(* CODESYS project zamek.project

Project tree, tasks and I/O mapping:
  Device : CODESYS Control Win V3, 3S - Smart Software Solutions GmbH, order no. 305021, version 3.5.8.10
    application Application
      libraries: Standard, * (System)
      task MainTask (cyclic, interval t#20ms, priority 1) calls PLC_PRG
      task VISU_TASK (cyclic, interval 100 ms, priority 31) calls VisuElems.Visu_Prg
      program PLC_PRG [ST]
      visualisation Visualization
  libraries: VisuSymbols, 3.5.8.0 (System)
  text list GlobalTextList
*)

// Device/Application/PLC_PRG
PROGRAM PLC_PRG

VAR								// Początek sekcji zmiennych
	
	xPrzycisk0: BOOL := FALSE;		// Zmienna stanu przycisku z cyfrą 0 (typ przycisku "pushswitch")	-> Zainicjalizowana wartością "false"
	xPrzycisk1: BOOL := FALSE;		// Zmienna stanu przycisku z cyfrą 1 (typ przycisku "pushswitch")	-> Zainicjalizowana wartością "false"	
	xPrzycisk2: BOOL := FALSE;		// Zmienna stanu przycisku z cyfrą 2 (typ przycisku "pushswitch")	-> Zainicjalizowana wartością "false"	
	xPrzycisk3: BOOL := FALSE;		// Zmienna stanu przycisku z cyfrą 3 (typ przycisku "pushswitch")	-> Zainicjalizowana wartością "false"	
	xPrzycisk4: BOOL := FALSE;		// Zmienna stanu przycisku z cyfrą 4 (typ przycisku "pushswitch")	-> Zainicjalizowana wartością "false"	
	xPrzycisk5: BOOL := FALSE;		// Zmienna stanu przycisku z cyfrą 5 (typ przycisku "pushswitch")	-> Zainicjalizowana wartością "false"	
	xPrzycisk6: BOOL := FALSE;		// Zmienna stanu przycisku z cyfrą 6 (typ przycisku "pushswitch")	-> Zainicjalizowana wartością "false"	
	xPrzycisk7: BOOL := FALSE;		// Zmienna stanu przycisku z cyfrą 7 (typ przycisku "pushswitch")	-> Zainicjalizowana wartością "false"	
	xPrzycisk8: BOOL := FALSE;		// Zmienna stanu przycisku z cyfrą 8 (typ przycisku "pushswitch")	-> Zainicjalizowana wartością "false"	
	xPrzycisk9: BOOL := FALSE;		// Zmienna stanu przycisku z cyfrą 9 (typ przycisku "pushswitch")	-> Zainicjalizowana wartością "false"	
	
	xKlucz: BOOL;					// Zmienna stanu przycisku typu "PowerSwitch" o nazwie "klucz"	
	xLampka1: BOOL;					// Zmienna oznaczająca stan lampki zielonej (typ "lamp1") - zapala się po wprowadzeniu prawidłowej sekwencji 4 cyfr
	xLampka2: BOOL;					// Zmienna oznaczająca stan lampki czerwonej (typ "lamp1") - zapala się po wprowadzeniu nieprawidłowej sekwencji cyfr
	
	xSpr1: BOOL;					// Zmienna typu "BOOL" oznaczająca wystukanie pierwszej poprawnej cyfry
	xSpr2: BOOL;					// Zmienna typu "BOOL" oznaczająca wystukanie drugiej poprawnej cyfry (1 cyfra poprawna musi być wprowadzona) 
	xSpr3: BOOL;					// Zmienna typu "BOOL" oznaczająca wystukanie trzeciej poprawnej cyfry (1 i 2 cyfra poprawna muszą być wprowadzone) 
	xSpr4: BOOL;					// Zmienna typu "BOOL" oznaczająca wystukanie czwartej poprawnej cyfry (1 i 2 i 3 cyfra poprawna muszą być wprowadzone)

	xOdblokuj: BOOL;				// Zmienna true/false zapalająca się (stan wysoki) jeśli cyfry poprawne zostały wprowadzone w prawidłowej sekwencji oraz oprócz tego czy przycisk "xKlucz" jest aktywny
	T3: TON;						// Deklaracja bloku funkcji Timer on-delay, który przeprowadza opóźnienie załączania stanu wysokiego w zmiennej "xOdblokuj2". Wynika z przyjętego algorytmu - ustawione opóźnienie jest niezauważalne
	xOdblokuj2: BOOL;				// Zmienna przyjmująca stan wysoki po upływie 1ms od ustawienia stanu wyokiego na zmiennej xOdblokuj 
	T1: TOF;						// Deklaracja bloku funkcji Timer off-delay przeprowadzającego opóźnienie wyłączenia lampki zielonej (xLampka1) - po 5s. Startuje swoje działanie, jeżeli zmienna xOdblokuj osiągnie opadające zbocze
	
	xNieOdblokuj: BOOL;				// Zmienna do obsługi wprowadzonego nieprawidłowego kodu / sekwencji. Osiąga stan wysoki jeżeli xKlucz osiąga stan wysoki, ale któraś ze zmiennych spr1,spr2,spr3,spr4 ma ustawiony stan niski
	T4: TON;						// Timer opóżniający zapalenie stanu wysokiego na zmiennej xNieOdblokuj2 o 1ms. Wynika z przyjętego algorytmu - ustawione opóźnienie jest niezauważalne.
	xNieOdblokuj2: BOOL;			// Zapala sie poprzez Timer po upłynięciu 1ms stanu wysokiego na zmiennej xNieOdblokuj		
	T2: TOF;						// Timer, który przy stanie niski zmiennej xNieOdblokuj załącza lampke czerwoną na 10s
	

	xNieaktywny: BOOL := FALSE;		// Zmienna służąca do poinformowaniu o bezczynności przycisku 'klucz' jeżeli któraś z lampek jest zapalona. Jest pezpośrednio podłączona do "xKlucz" powershitch do wejścia "deactivate inputs" w wizualizacji (powerswitch properties)
	
	xLicznikProb1: INT := 0;		// Licznik nieudanych prób. Jest zwiększany o 2 przy każdej nieudanej próbie (przy sprawdzaniu spr1,spr2,spr3,spr4 oraz zKlucz). Kiedy osiąga wartość 6 - 3 nieudane próby - następuje załączenie lampki czerwonej na 3min.
	
	xBlokuj: BOOL := FALSE;			// Jest odpowiednikiem xNieOdblokuj - stworzona w celu obsługi trzyminutowego zapalenia czerwonej lampki. Stworzona na potrzeby przyjętego algorytmu - 'steruje' zmienną xBlokuj2
	xBlokuj2: BOOL := FALSE;		// Jest odpowiednikiem xNieOdblokuj2 - stworzona w celu obsługi trzyminutowego zapalenia czerwonej lampki. Jej stan niski powoduje opóźnienie (zapalenia lampki czerwonej) na 3min
	
	T5: TOF;						// Odpowiednik Timera T2, który odpowiada za bezpośrednie ustawienie stanu wysokiego na lampce czerwonej na 3min
	T6: TON;						// Odpowiednik Timera T4, który po upływie 1ms ustawia stan niski na xBlokuj2
	
	xZerujLIcznik2: BOOL := FALSE;	// Zmienna stworzona do sprawdzania liczby prób (xLiczbProb1). Przyjmuje stan wysoki jeżeli 3 próba z kolei się nie powiodła 
	xZerujLIcznik: BOOL := FALSE;	// Zapala się tutaj stan wysoki po upłynięciu 3 min od zapalenia stanu wysokiego na zmiennej xZerujLicznik2. Te dwie zmienne sterują prawidłowym procesem zerowania liczby prób po upływie 3 minut - 3 nieudane próby
	T7: TON;						// Blok Timer, który ustawia stan wysoki na zmiennej xZerujLIcznik po upłynięciu 3 min ustawienia lampki czerwonej - stanu wysokiego na zmiennej xZerujLicznik2
	
END_VAR							// Koniec sekcji zmiennych

// Sekcja właściwego kodu programu

	// KOD POPRAWNY DO OTWORZENIA ZAMKA: 1234
	// KOD POPRAWNY DO OTWORZENIA ZAMKA: 1234
	// KOD POPRAWNY DO OTWORZENIA ZAMKA: 1234
	
	// Sprawdzanie prawidłowej sekwencji oraz prawidłowych cyfr zamka
	
		// Czy przycisk z cyfrą 1 został naciśnięty - żadne inne
		
			IF (xPrzycisk0=FALSE AND xPrzycisk5=FALSE AND xPrzycisk6=FALSE AND xPrzycisk7=FALSE AND xPrzycisk8=FALSE AND xPrzycisk9=FALSE) AND xPrzycisk1=TRUE AND xPrzycisk2=FALSE AND xPrzycisk3=FALSE AND xPrzycisk4=FALSE AND xKlucz=FALSE THEN
				xSpr1:=TRUE;
			END_IF

		// Czy przycisk z cyfrą 2 został naciśnięty (i przycisk z cyfrą 1 jest dalej aktywny) - żadne inne
			
			IF (xPrzycisk0=FALSE AND xPrzycisk5=FALSE AND xPrzycisk6=FALSE AND xPrzycisk7=FALSE AND xPrzycisk8=FALSE AND xPrzycisk9=FALSE) AND xPrzycisk2=TRUE AND xPrzycisk3=FALSE AND xPrzycisk4=FALSE AND xSpr1=TRUE AND xKlucz=FALSE THEN
				xSpr2:=TRUE;
			END_IF
			
		// Czy przycisk z cyfrą 3 został naciśnięty (i przycisk z cyfrą 1 i 2 jest dalej aktywny) - żadne inne

			IF (xPrzycisk0=FALSE AND xPrzycisk5=FALSE AND xPrzycisk6=FALSE AND xPrzycisk7=FALSE AND xPrzycisk8=FALSE AND xPrzycisk9=FALSE) AND xPrzycisk3=TRUE AND xPrzycisk4=FALSE AND xSpr1=TRUE AND xSpr2=TRUE AND xKlucz=FALSE THEN
				xSpr3:=TRUE;
			END_IF
			
		// Jeżeli został wciśnięty inny przycisk to zmienna określająca wysoki stan na przycisku 1 2 3 zmienia się na false - zapobiegnięcie m.in. sytuacji kodu 1 2 3 4 5

			IF (xPrzycisk5=TRUE OR xPrzycisk6=TRUE OR xPrzycisk7=TRUE OR xPrzycisk8=TRUE OR xPrzycisk9=TRUE) THEN
				xSpr3:=FALSE;
			END_IF
			
		// Czy przycisk z cyfrą 4 został naciśnięty (i przycisk z cyfrą 1 i 2 i 3 jest dalej aktywny) - żadne inne

			IF (xPrzycisk0=FALSE AND xPrzycisk5=FALSE AND xPrzycisk6=FALSE AND xPrzycisk7=FALSE AND xPrzycisk8=FALSE AND xPrzycisk9=FALSE) AND xPrzycisk4=TRUE AND xSpr1=TRUE AND xSpr2=TRUE AND xSpr3=TRUE AND xKlucz=FALSE THEN
				xSpr4:=TRUE;
			END_IF
		
		// Sekwencja 1 2 3 4 ustawia stan wysoki na zmiennej xOdblokuj (zaraz po naciśnięciu przycisku klucz)
			
			IF xSpr1=TRUE AND xSpr2=TRUE AND xSpr3=TRUE AND xSpr4=TRUE AND xKlucz=TRUE THEN
				xOdblokuj:=TRUE;
			END_IF

		// Kod wynikający z opracowanego algorytmu. Zmiana stanu zmainnej xOdblokuj2 (na wysoki) pod wpływem ustawienia stanu wysokiego xOdblokuj po 1ms 	
			
			T3(IN:=xOdblokuj,PT:=T#1MS);		// Deklaracja Timera TON. IN-zmienna wejściowa, PT-czas do ustawienia zmiennej wyjściowej
			xOdblokuj2:=T3.Q;					// Poinformowanie o zmiennej wyjściowej

		// Kod poniżej wykouje się w przypadku prawidłowej sekwencji. Wszystkie potrzebne przyciski, zmienne sprawdzające, licznik nieudanych prób, zostają "zresetowane" - ustawione na stan niski	
			
			IF xOdblokuj2=TRUE THEN
				xOdblokuj:=FALSE;
				
				xSpr1:=FALSE;
				xSpr2:=FALSE;
				xSpr3:=FALSE;
				xSpr4:=FALSE;
				
				xKlucz:=FALSE;
				xPrzycisk0:=FALSE;	
				xPrzycisk1:=FALSE;	
				xPrzycisk2:=FALSE;
				xPrzycisk3:=FALSE;
				xPrzycisk4:=FALSE;
				xPrzycisk5:=FALSE;
				xPrzycisk6:=FALSE;
				xPrzycisk7:=FALSE;
				xPrzycisk8:=FALSE;
				xPrzycisk9:=FALSE;
				
				xBlokuj:=FALSE;
				xBlokuj2:=FALSE;
				
				xLicznikProb1:=0;		// licznik nieudanych prób zeruje się, gdzy wprowadzono prawidłową sekwencję cyfr
			END_IF

		//	Obsługa załączenie lampki czerwonej na 5s w przypadku udanej próby otwarcia zamka pod wpływem ustawienia stanu niskiego w zmiennej xOdblokuj
		
			T1(IN:=xOdblokuj,PT:=T#5S);
			xLampka1:=T1.Q;

	//	Instrukcje warunkowe obsługujące zerowanie licznika prób, gdy nastąpiło już 3 minutowe zapalenie czerwonej lampki

		IF xZerujLIcznik=TRUE THEN
			xLicznikProb1:=0;
		END_IF

		IF xLicznikProb1=0 THEN
			xZerujLIcznik:=FALSE;
			xZerujLIcznik2:=FALSE;
		END_IF
		
	//	Obsługa wprowadzenia nieprawidłowego kodu

		IF (xSpr1=FALSE OR xSpr2=FALSE OR xSpr3=FALSE OR xSpr4=FALSE) AND xKlucz=TRUE THEN
			xNieOdblokuj:=TRUE;					// aby czerwona lampka zaświeciła się na 10s
			xBlokuj:=TRUE;						// aby czerwona lampka zaświeciła się na 3min
			xLicznikProb1:=xLicznikProb1+1;		// licznik nieudanych prób jest zwiększany o 2 - wartość 6 (3 nieudane próby) to załączenie lampki czerwonej i nieaktywność zamka na 3 min
		END_IF

		
	// Obsługa Timerów TON
	
		T6(IN:=xBlokuj,PT:=T#1MS);			// 1ms - wynika z wymyślonego algorytmu. Zmiana potrzebnej wartości typu bool
		xBlokuj2:=T6.Q;

		T4(IN:=xNieOdblokuj,PT:=T#1MS);		// 1ms - wynika z wymyślonego algorytmu. Zmiana potrzebnej wartości typu bool
		xNieOdblokuj2:=T4.Q;

	// Poniższy kod dla nieaktywności zamka przez 3min. Nieudane próbny = 3	(xLicznikProb1 = 6)
		
		IF xNieOdblokuj2=TRUE AND xBlokuj2=TRUE AND xLicznikProb1=6 THEN
			xBlokuj:=FALSE;			// Następstwem tej zmiany stanu jest wywołanie timera na 180s
			xSpr1:=FALSE;
			xSpr2:=FALSE;
			xSpr3:=FALSE;
			xSpr4:=FALSE;
			xKlucz:=FALSE;
			xPrzycisk0:=FALSE;	
			xPrzycisk1:=FALSE;	
			xPrzycisk2:=FALSE;
			xPrzycisk3:=FALSE;
			xPrzycisk4:=FALSE;
			xPrzycisk5:=FALSE;
			xPrzycisk6:=FALSE;
			xPrzycisk7:=FALSE;
			xPrzycisk8:=FALSE;
			xPrzycisk9:=FALSE;
		END_IF

	// Poniższy kod dla nieaktywności zamka przez tylko 10s	- liczba nieudanych prób różna od 3 (czyli xLicznikProb1 <> 6)	
		
		IF xNieOdblokuj2=TRUE AND xLicznikProb1<>6 THEN
			xNieOdblokuj:=FALSE;		// Następstwem tej zmiany stanu jest wywołanie timera na 10s
			xSpr1:=FALSE;
			xSpr2:=FALSE;
			xSpr3:=FALSE;
			xSpr4:=FALSE;
			xKlucz:=FALSE;
			xPrzycisk0:=FALSE;	
			xPrzycisk1:=FALSE;	
			xPrzycisk2:=FALSE;
			xPrzycisk3:=FALSE;
			xPrzycisk4:=FALSE;
			xPrzycisk5:=FALSE;
			xPrzycisk6:=FALSE;
			xPrzycisk7:=FALSE;
			xPrzycisk8:=FALSE;
			xPrzycisk9:=FALSE;
		END_IF

	// Załączenie lampki czerwonej na 180s, gdy zmienna xBlokuj będzie w stanie niskim 
											// Timer TOF
		T5(IN:=xBlokuj,PT:=T#180S);			// opadające zbocze xBlokuj startuje Timer na 180s
		xLampka2:=T5.Q;						// Zmienna wyjściowa
		
	// Załączenie lampki czerwonej na 10s, gdy zmienna xNieOdblokuj będzie w stanie niskim 	
											// Timer TOF
		T2(IN:=xNieOdblokuj,PT:=T#10S);		// opadające zbocze xNieOdblokuj startuje Timer na 10s
		xLampka2:=T2.Q;						// Zmienna wyjściowa


	//	Instrukcja warunkowa dla niekatywności przycisku klucza - "powerswitch" w wizualizacji

		IF xLampka1=TRUE OR xLampka2=TRUE THEN	// jeżeli któraś z lampek świeci
			xNieaktywny:=TRUE;					// ta zmienna jest przypisana do dezaktywacji przycisku xKlucz
		END_IF

	//	Instrukcja warunkowa poniżej została stworzona w celu ustawienia stanu wyskoiego na zmiennej xZerujLIcznik2, czego następstwem będzie uruchomienia Timera TON 
		
		IF xNieaktywny=TRUE AND xLicznikProb1>=6 THEN
			xPrzycisk0:=FALSE;	
			xPrzycisk1:=FALSE;	
			xPrzycisk2:=FALSE;
			xPrzycisk3:=FALSE;
			xPrzycisk4:=FALSE;
			xPrzycisk5:=FALSE;
			xPrzycisk6:=FALSE;
			xPrzycisk7:=FALSE;
			xPrzycisk8:=FALSE;
			xPrzycisk9:=FALSE;
			xBlokuj:=FALSE;
			xBlokuj2:=FALSE;
			xZerujLIcznik2:=TRUE;
		END_IF;
		
	// Timer TON (poniżej) startujący poprzez ustawienie zmiennej xZerujLIcznik2 na stan wysoki w poprzedniej instrukcji warunkowej. Stworzony w celu prawidłowego działania lampki czerwonej dla 3 minut jej zapalenia

		T7(IN:=xZerujLIcznik2,PT:=T#180S);
		xZerujLIcznik:=T7.Q;				// Po upływie 3min (lampka czerwona gaśnie). Ustawiany jest stan wysoki na zmiennej xZerujLIcznik. Ta zmienna jest sprawdzana na początku programu. Jej stan wysoki tam powoduje bezpośrdnie wyzerowanie zmiennej typu int z liczbą nieudanych prób

	// gdy przycisk xKlucz będzie nieaktywny inne przyciski będą ustawione w stan niski

		IF xNieaktywny=TRUE THEN
			xPrzycisk0:=FALSE;	
			xPrzycisk1:=FALSE;	
			xPrzycisk2:=FALSE;
			xPrzycisk3:=FALSE;
			xPrzycisk4:=FALSE;
			xPrzycisk5:=FALSE;
			xPrzycisk6:=FALSE;
			xPrzycisk7:=FALSE;
			xPrzycisk8:=FALSE;
			xPrzycisk9:=FALSE;
			xBlokuj:=FALSE;
			xBlokuj2:=FALSE;
		END_IF;

	// aktywacja przycisku xKlucz poprzez zmienną xNieaktywny ustawioną na false - xKlucz properties w visualization - deactivate inputs

		IF xLampka1=FALSE AND xLampka2=FALSE THEN
			xNieaktywny:=FALSE;
		END_IF;

// Koniec sekcji właściwego kodu programu

END_PROGRAM

// Device/Application/Visualization
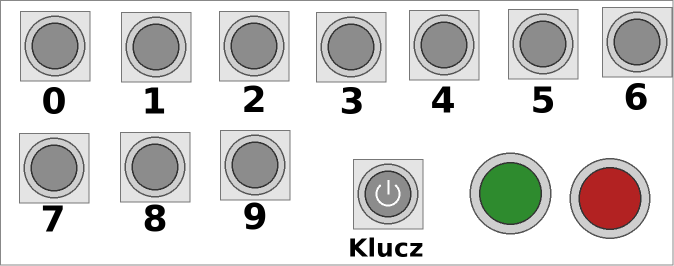
VISUALIZATION Visualization  // 674x266
    PushSwitch (121,12 70x70), variable: PLC_PRG.xPrzycisk1, behaviour: TOGGLE, style: Switch-PushSwitch-Gray
    PushSwitch (219,11 70x70), variable: PLC_PRG.xPrzycisk2, behaviour: TOGGLE, style: Switch-PushSwitch-Gray
    PushSwitch (316,12 70x70), variable: PLC_PRG.xPrzycisk3, behaviour: TOGGLE, style: Switch-PushSwitch-Gray
    PushSwitch (409,10 70x70), variable: PLC_PRG.xPrzycisk4, behaviour: TOGGLE, style: Switch-PushSwitch-Gray
    Label (131,84 46x34), "1"
    PushSwitch (508,9 70x70), variable: PLC_PRG.xPrzycisk5, behaviour: TOGGLE, style: Switch-PushSwitch-Gray
    PushSwitch (602,7 70x70), variable: PLC_PRG.xPrzycisk6, behaviour: TOGGLE, style: Switch-PushSwitch-Gray
    PushSwitch (120,132 70x70), variable: PLC_PRG.xPrzycisk8, behaviour: TOGGLE, style: Switch-PushSwitch-Gray
    PushSwitch (19,133 70x70), variable: PLC_PRG.xPrzycisk7, behaviour: TOGGLE, style: Switch-PushSwitch-Gray
    PushSwitch (220,130 70x70), variable: PLC_PRG.xPrzycisk9, behaviour: TOGGLE, style: Switch-PushSwitch-Gray
    Label (30,204 46x30), "7"
    Label (613,80 46x34), "6"
    Label (231,81 46x37), "2"
    Label (329,84 46x34), "3"
    Label (520,83 46x34), "5"
    Label (420,85 46x30), "4"
    Label (132,201 46x35), "8"
    Label (232,200 46x33), "9"
    Label (323,231 126x33), "Klucz"
    Lamp1 (563,147 94x103), variable: PLC_PRG.xLampka2, style: Lamp-Lamp1-Red
    Lamp1 (461,146 99x95), variable: PLC_PRG.xLampka1, style: Lamp-Lamp1-Green
    PushSwitch (20,11 70x70), variable: PLC_PRG.xPrzycisk0, behaviour: TOGGLE, style: Switch-PushSwitch-Gray
    Label (31,84 46x34), "0"
    PowerSwitch (353,159 70x70), variable: PLC_PRG.xKlucz, input disabled if: PLC_PRG.xNieaktywny, behaviour: TOGGLE, style: Switch-PowerSwitch-Gray
END_VISUALIZATION
